Staubli VAL3: ros_i_driver.pjx

--- ros_i_driver.pjx ---
Parameters version=s7.7.2 stackSize=5000 millimeterUnit=true
Program file=encodeJointFbk.pgx
Program file=encodeJState.pgx
Program file=encodeStatus.pgx
Program file=fbkStreamer.pgx
Program file=initParams.pgx
Program file=jStateStreamer.pgx
Program file=sendJointFbk.pgx
Program file=sendJState.pgx
Program file=setupRosMsgs.pgx
Program file=start.pgx
Program file=stop.pgx
Data file=ros_i_driver.dtx
Type name=RosSimpleMsg path=Disk://RosSimpleMsg/RosSimpleMsg.pjx

--- ros_i_driver.dtx ---
public bool bFbkOverrun
public bool bMotionOverrun
public jointRx jCurrPose
mdesc mNomSpeed = {blend=off}
public num nCounter
public num nFbkPeriod = 0.032
public num nLengthB[4]
num nMotionPeriod = 0.012
public num nPosVelAccB[120]
public num nRetVal
public num nRobotIdB[4]
public num nTimeB[4]
public num nValidFieldsB[4] = 2
public sio siTcpIpFbk = {link=Socket\Feedback}
public sio siTcpIpMotion = {link=Socket\Motion}
public string sFbkTaskName = "publisher"
public string sMotionTaskName
public num nMsgTypeB[4]
public num nCommTypeB[4]
public num nReplyCodeB[4]
public RosSimpleMsg rosMsgJointFbk
  [0]
    Header header
      [0]
        num nMsgType
        num nCommType
        num nReplyCode
    Prefix prefix
      [0]
        num nLength
    Body body
      [0]
        num nData[33]
public bool bStream
public num nBytesSent
public RosSimpleMsg rosMsgJState
  [0]
    Header header
      [0]
        num nMsgType
        num nCommType
        num nReplyCode
    Prefix prefix
      [0]
        num nLength
    Body body
      [0]
        num nData[11]
public num nSeqB[4]
public num nPosB[40]
public num nDeg2Rad

--- start.pgx ---
program start()
begin
  userPage()
  cls()

  // feedback task will run every 32 ms (approx. 31 HZ)
  //nFbkPeriod=0.032
  nFbkPeriod=0.05
  // motion task will run every 12 ms (approx. 83 Hz)
  nMotionPeriod=0.012

  nDeg2Rad = 3.14159265359 / 180.0

  sFbkTaskName="publisher"

  // initialise TCP/IP parameters
  //call initParams()

  // create feedback (state and status) task to send data to industrial_robot)client
  taskCreateSync sFbkTaskName,nFbkPeriod,bFbkOverrun,jStateStreamer()

end

--- encodeJointFbk.pgx ---
public program encodeJointFbk()
begin
  // encode prefix length
  nRetVal=toBinary(rosMsgJointFbk.prefix.nLength, 1, "-4l", nLengthB)

  // encode header
  nRetVal=toBinary(rosMsgJointFbk.header.nMsgType, 1, "-4l", nMsgTypeB)
  nRetVal=toBinary(rosMsgJointFbk.header.nCommType, 1, "-4l", nCommTypeB)
  nRetVal=toBinary(rosMsgJointFbk.header.nReplyCode, 1, "-4l", nReplyCodeB)

  // encode first 3 variables of body message (data)
  nRetVal=toBinary(rosMsgJointFbk.body.nData, 1, "-4l", nRobotIdB)
  nRetVal=toBinary(rosMsgJointFbk.body.nData[1], 1, "-4l", nValidFieldsB)
  nRetVal=toBinary(rosMsgJointFbk.body.nData[2], 1, "4.0l", nTimeB)

  // assuming the remaining elements have zeros assigned by default
  rosMsgJointFbk.body.nData[3] = jCurrPose.j1
  rosMsgJointFbk.body.nData[4] = jCurrPose.j2
  rosMsgJointFbk.body.nData[5] = jCurrPose.j3
  rosMsgJointFbk.body.nData[6] = jCurrPose.j4
  rosMsgJointFbk.body.nData[7] = jCurrPose.j5
  rosMsgJointFbk.body.nData[8] = jCurrPose.j6

  // encode 30 values representing Positions[10], Velocities[10] and Accelerations[10]
  nRetVal=toBinary(rosMsgJointFbk.body.nData[3], 30, "4.0l", nPosVelAccB)
end

--- encodeJState.pgx ---
public program encodeJState()
begin
  // encode prefix length
  nRetVal=toBinary(rosMsgJointFbk.prefix.nLength, 1, "-4l", nLengthB)

  // encode header
  nRetVal=toBinary(rosMsgJointFbk.header.nMsgType, 1, "-4l", nMsgTypeB)
  nRetVal=toBinary(rosMsgJointFbk.header.nCommType, 1, "-4l", nCommTypeB)
  nRetVal=toBinary(rosMsgJointFbk.header.nReplyCode, 1, "-4l", nReplyCodeB)

  // encode 'sequence' variable of body message (data)
  nRetVal=toBinary(rosMsgJointFbk.body.nData, 1, "-4l", nSeqB)

  // assuming the remaining elements have zeros assigned by default
  rosMsgJState.body.nData[1] = jCurrPose.j1 * nDeg2Rad
  rosMsgJState.body.nData[2] = jCurrPose.j2 * nDeg2Rad
  rosMsgJState.body.nData[3] = jCurrPose.j3 * nDeg2Rad
  rosMsgJState.body.nData[4] = jCurrPose.j4 * nDeg2Rad
  rosMsgJState.body.nData[5] = jCurrPose.j5 * nDeg2Rad
  rosMsgJState.body.nData[6] = jCurrPose.j6 * nDeg2Rad

  // encode 10 values representing joints[10]
  nRetVal=toBinary(rosMsgJState.body.nData[1], 10, "4.0l", nPosB)
end

--- encodeStatus.pgx ---
public program encodeStatus()
begin
end

--- fbkStreamer.pgx ---
public program fbkStreamer()
begin
  bStream = true
  call setupRosMsgs()
  while (bStream)
    // fetch robot status
    //call fetchStatus()

    // encode and send ROS simple message ID 13: robot status
    //call encodeStatus()
    //call sendRosMsg(rosMsgStatus)

    // fetch current joint values
    jCurrPose=herej()

    // encode and send ROS simple_message ID 15: joint feedback
    call encodeJointFbk()
    nBytesSent = 0
    call sendJointFbk()
    delay(0)
  endWhile
end

--- initParams.pgx ---
public program initParams()
begin
  nRetVal=sioCtrl(siTcpIpFbk,"port",11002)
  if (nRetVal!=0)
    popUpMsg("Error while setting IP port")
    //return ?
  endIf

  nRetVal=sioCtrl(siTcpIpFbk,"timeout",5)
  if (nRetVal!=0)
    popUpMsg("Error while setting TCP/IP timeout")
    //return ?
  endIf
end

--- jStateStreamer.pgx ---
public program jStateStreamer()
begin
  bStream = true
  call setupRosMsgs()
  while (bStream)
    // fetch robot status
    //call fetchStatus()

    // encode and send ROS simple message ID 13: robot status
    //call encodeStatus()
    //call sendRosMsg(rosMsgStatus)

    // fetch current joint values
    jCurrPose=herej()

    // encode and send ROS simple_message ID 15: joint feedback
    call encodeJState()
    nBytesSent = 0
    call sendJState()
    delay(0)
  endWhile
end

--- sendJointFbk.pgx ---
public program sendJointFbk()
begin
  // send message length (prefix)
  nRetVal = sioSet(siTcpIpFbk, nLengthB)
  if (nRetVal == -1)
    putln("Client not connected")
    return
  elseIf (nRetVal < 4)
    popUpMsg("Error while sending prefix")
  endIf

  nBytesSent = size(nLengthB)

  // send message header (msg type, comm type, reply code)
  nRetVal = sioSet(siTcpIpFbk, nMsgTypeB)
  if (nRetVal == -1)
    putln("Client disconnected")
    bStream = false
    return
  elseIf (nRetVal < 4)
    popUpMsg("Error while sending msg type")
  endIf

  nBytesSent = nBytesSent + size(nMsgTypeB)

  nRetVal = sioSet(siTcpIpFbk, nCommTypeB)
  if (nRetVal == -1)
    putln("Client disconnected")
    bStream = false
    return
  elseIf (nRetVal < 4)
    popUpMsg("Error while sending comm type")
  endIf

  nBytesSent = nBytesSent + size(nCommTypeB)

  nRetVal = sioSet(siTcpIpFbk, nReplyCodeB)
  if (nRetVal == -1)
    putln("Client disconnected")
    bStream = false
    return
  elseIf (nRetVal < 4)
    popUpMsg("Error while sending reply code")
  endIf

  nBytesSent = nBytesSent + size(nReplyCodeB)

  // send message body (data)
  // send robotId
  nRetVal = sioSet(siTcpIpFbk, nRobotIdB)
  if (nRetVal == -1)
    putln("client disconnected")
    bStream = false
    return
  elseIf (nRetVal < 4)
    popUpMsg("Error while sending robot ID")
  endIf

  nBytesSent = nBytesSent + size(nRobotIdB)

  // send validFields
  nRetVal = sioSet(siTcpIpFbk, nValidFieldsB)
  if (nRetVal == -1)
    putln("client disconnected")
    bStream = false
    return
  elseIf (nRetVal < 4)
    popUpMsg("Error while sending valid fields")
  endIf

  nBytesSent = nBytesSent + size(nValidFieldsB)

  // send Time
  nRetVal = sioSet(siTcpIpFbk, nTimeB)
  if (nRetVal == -1)
    putln("client disconnected")
    bStream = false
    return
  elseIf (nRetVal < 4)
    popUpMsg("Error while sending timestamp")
  endIf

  nBytesSent = nBytesSent + size(nTimeB)

  // send positions[], velocities[] and accelerations[]
  nRetVal = sioSet(siTcpIpFbk, nPosVelAccB)
  if (nRetVal == -1)
    putln("Client disconnected")
    bStream = false
    return
  elseIf (nRetVal < size(nPosVelAccB))
    popUpMsg("Error while sending msg body")
  endIf

  nBytesSent = nBytesSent + size(nPosVelAccB)

  //put("Joint status sent: ")
  //putln(nBytesSent)
  //bStream = false
end

--- sendJState.pgx ---
public program sendJState()
begin
  // send message length (prefix)
  nRetVal = sioSet(siTcpIpFbk, nLengthB)
  if (nRetVal == -1)
    putln("Client not connected")
    return
  elseIf (nRetVal < 4)
    popUpMsg("Error while sending prefix")
  endIf

  nBytesSent = size(nLengthB)

  // send message header (msg type, comm type, reply code)
  nRetVal = sioSet(siTcpIpFbk, nMsgTypeB)
  if (nRetVal == -1)
    putln("Client disconnected")
    bStream = false
    return
  elseIf (nRetVal < 4)
    popUpMsg("Error while sending msg type")
  endIf

  nBytesSent = nBytesSent + size(nMsgTypeB)

  nRetVal = sioSet(siTcpIpFbk, nCommTypeB)
  if (nRetVal == -1)
    putln("Client disconnected")
    bStream = false
    return
  elseIf (nRetVal < 4)
    popUpMsg("Error while sending comm type")
  endIf

  nBytesSent = nBytesSent + size(nCommTypeB)

  nRetVal = sioSet(siTcpIpFbk, nReplyCodeB)
  if (nRetVal == -1)
    putln("Client disconnected")
    bStream = false
    return
  elseIf (nRetVal < 4)
    popUpMsg("Error while sending reply code")
  endIf

  nBytesSent = nBytesSent + size(nReplyCodeB)

  // send message body (data)
  // send sequence
  nRetVal = sioSet(siTcpIpFbk, nSeqB)
  if (nRetVal == -1)
    putln("client disconnected")
    bStream = false
    return
  elseIf (nRetVal < 4)
    popUpMsg("Error while sending sequence")
  endIf

  nBytesSent = nBytesSent + size(nSeqB)

  // send joints[]
  nRetVal = sioSet(siTcpIpFbk, nPosB)
  if (nRetVal == -1)
    putln("Client disconnected")
    bStream = false
    return
  elseIf (nRetVal < size(nPosB))
    popUpMsg("Error while sending msg body")
  endIf

  nBytesSent = nBytesSent + size(nPosB)

  //put("Joint state sent: ")
  //putln(nBytesSent)
  //bStream = false
end

--- setupRosMsgs.pgx ---
public program setupRosMsgs()
begin
  // Robot status message
  //rosMsgStatus.header.nMsgType=13
  //rosMsgStatus.header.nCommType=1
  //rosMsgStatus.header.nReplyCode=0

  // Joint trajectory point message
  //rosMsgJointTraj.header.nMsgType=14
  //rosMsgJointTraj.header.nCommType=1
  //rosMsgJointTraj.header.nReplyCode=0

  // Feedback of joint position/velocity/acceleration
  // prefix length = 12 + 132 = 144
  //rosMsgJointFbk.prefix.nLength=144
  //rosMsgJointFbk.header.nMsgType=15
  //rosMsgJointFbk.header.nCommType=1
  //rosMsgJointFbk.header.nReplyCode=0

  // robot_id
  //rosMsgJointFbk.body.nData[0] = 0
  // valid_fields
  //rosMsgJointFbk.body.nData[1] = 2
  // time
  //rosMsgJointFbk.body.nData[2] = 3.2


  // Feedback of joint position
  // prefix length = 12 + 44
  rosMsgJointFbk.prefix.nLength=56
  rosMsgJointFbk.header.nMsgType=10
  rosMsgJointFbk.header.nCommType=1
  rosMsgJointFbk.header.nReplyCode=0
  // sequence
  rosMsgJointFbk.body.nData[0] = 0
end

--- stop.pgx ---
program stop()
begin
  resetMotion()
  popUpMsg("Pending movement commands have been cancelled.")
  cls()
end
